// TIA Portal V17 export
// export: Created 2025-03-05T08:03:01.8804451Z, ExportSetting WithDefaults, DisplayName Totally Integrated Automation Portal, DisplayVersion V17 Update 8, DisplayName TIA Portal Openness, DisplayVersion V17 Update 8, DisplayName TIA Portal Version Control Interface, DisplayVersion V17, DisplayName SINAMICS Startdrive Advanced, DisplayVersion V17 SP2, DisplayName SINAMICS Startdrive G110M, G120, G120C, G120D, G120P, G115D, DisplayVersion V17 SP2, DisplayName SINAMICS Startdrive G130, G150, S120, S150, SINAMICS MV, S210, DisplayVersion V17 SP2, DisplayName STEP 7 Professional, DisplayVersion V17 Update 8, DisplayName SINUMERIK ONE STEP 7 Toolbox, DisplayVersion V17 Update 12, DisplayName SINUMERIK 840D sl STEP 7 Toolbox, DisplayVersion V17 Update 12, DisplayName STEP 7 Safety, DisplayVersion V17 Update 6, DisplayName WinCC Advanced, DisplayVersion V17 Update 8
FUNCTION "FC21011_POWDER_FEEDER_GENERAL" : Void   // FC21011, LAD
TITLE = FC21011 POWDER FEEDER GENERAL
{ S7_Optimized_Access := 'TRUE' }
VERSION : 0.1
// stored: AutoNumber false, IsIECCheckEnabled false, SetENOAutomatically false, UDAEnableTagReadback false
BEGIN

REGION Network 1: /////_UNIT_01_/////
END_REGION

REGION Network 2: CALL FB21011 POWDER FEEDER 1 GENERAL UNIT 01
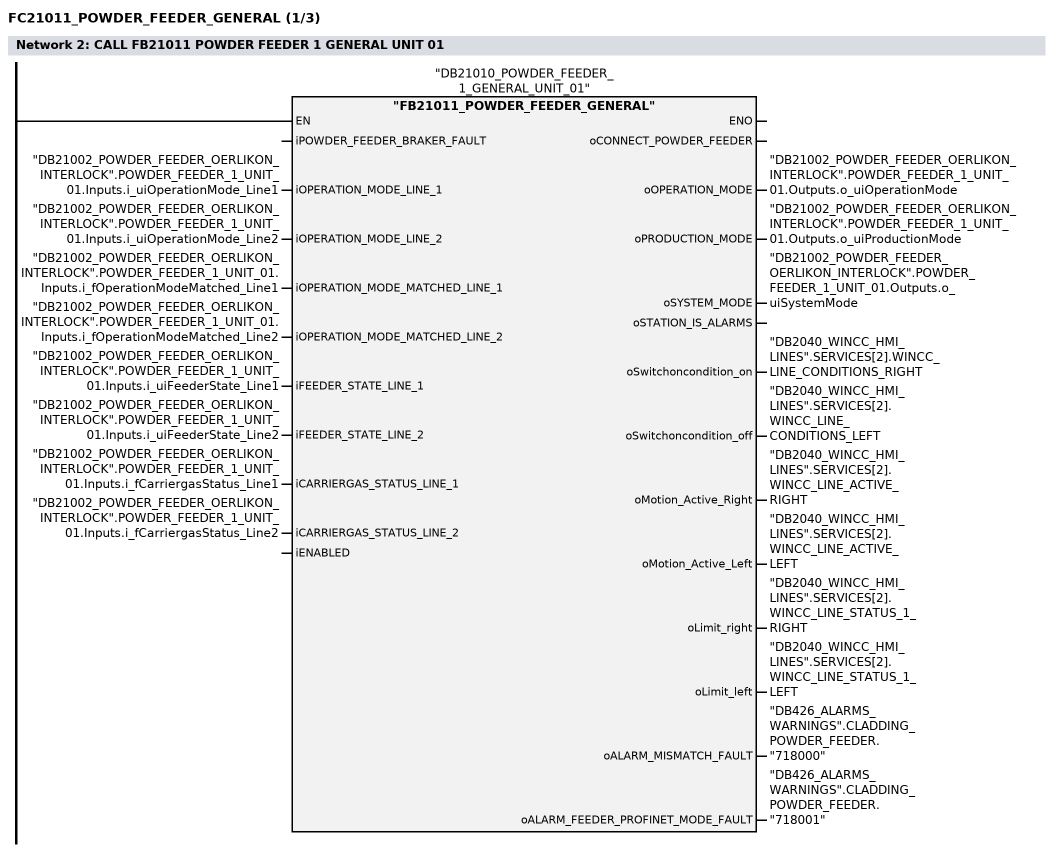
   RUNG wire#powerrail
      "DB21010_POWDER_FEEDER_1_GENERAL_UNIT_01"(iPOWDER_FEEDER_BRAKER_FAULT :=, iOPERATION_MODE_LINE_1 := "DB21002_POWDER_FEEDER_OERLIKON_INTERLOCK".POWDER_FEEDER_1_UNIT_01.Inputs.i_uiOperationMode_Line1, iOPERATION_MODE_LINE_2 := "DB21002_POWDER_FEEDER_OERLIKON_INTERLOCK".POWDER_FEEDER_1_UNIT_01.Inputs.i_uiOperationMode_Line2, iOPERATION_MODE_MATCHED_LINE_1 := "DB21002_POWDER_FEEDER_OERLIKON_INTERLOCK".POWDER_FEEDER_1_UNIT_01.Inputs.i_fOperationModeMatched_Line1, iOPERATION_MODE_MATCHED_LINE_2 := "DB21002_POWDER_FEEDER_OERLIKON_INTERLOCK".POWDER_FEEDER_1_UNIT_01.Inputs.i_fOperationModeMatched_Line2, iFEEDER_STATE_LINE_1 := "DB21002_POWDER_FEEDER_OERLIKON_INTERLOCK".POWDER_FEEDER_1_UNIT_01.Inputs.i_uiFeederState_Line1, iFEEDER_STATE_LINE_2 := "DB21002_POWDER_FEEDER_OERLIKON_INTERLOCK".POWDER_FEEDER_1_UNIT_01.Inputs.i_uiFeederState_Line2, iCARRIERGAS_STATUS_LINE_1 := "DB21002_POWDER_FEEDER_OERLIKON_INTERLOCK".POWDER_FEEDER_1_UNIT_01.Inputs.i_fCarriergasStatus_Line1, iCARRIERGAS_STATUS_LINE_2 := "DB21002_POWDER_FEEDER_OERLIKON_INTERLOCK".POWDER_FEEDER_1_UNIT_01.Inputs.i_fCarriergasStatus_Line2, iENABLED :=, oCONNECT_POWDER_FEEDER =>, oOPERATION_MODE => "DB21002_POWDER_FEEDER_OERLIKON_INTERLOCK".POWDER_FEEDER_1_UNIT_01.Outputs.o_uiOperationMode, oPRODUCTION_MODE => "DB21002_POWDER_FEEDER_OERLIKON_INTERLOCK".POWDER_FEEDER_1_UNIT_01.Outputs.o_uiProductionMode, oSYSTEM_MODE => "DB21002_POWDER_FEEDER_OERLIKON_INTERLOCK".POWDER_FEEDER_1_UNIT_01.Outputs.o_uiSystemMode, oSTATION_IS_ALARMS =>, oSwitchoncondition_on => "DB2040_WINCC_HMI_LINES".SERVICES[2].WINCC_LINE_CONDITIONS_RIGHT, oSwitchoncondition_off => "DB2040_WINCC_HMI_LINES".SERVICES[2].WINCC_LINE_CONDITIONS_LEFT, oMotion_Active_Right => "DB2040_WINCC_HMI_LINES".SERVICES[2].WINCC_LINE_ACTIVE_RIGHT, oMotion_Active_Left => "DB2040_WINCC_HMI_LINES".SERVICES[2].WINCC_LINE_ACTIVE_LEFT, oLimit_right => "DB2040_WINCC_HMI_LINES".SERVICES[2].WINCC_LINE_STATUS_1_RIGHT, oLimit_left => "DB2040_WINCC_HMI_LINES".SERVICES[2].WINCC_LINE_STATUS_1_LEFT, oALARM_MISMATCH_FAULT => "DB426_ALARMS_WARNINGS".CLADDING_POWDER_FEEDER."718000", oALARM_FEEDER_PROFINET_MODE_FAULT => "DB426_ALARMS_WARNINGS".CLADDING_POWDER_FEEDER."718001")
   END_RUNG
   // the same network as SCL:
   "DB21010_POWDER_FEEDER_1_GENERAL_UNIT_01"(iOPERATION_MODE_LINE_1 := "DB21002_POWDER_FEEDER_OERLIKON_INTERLOCK".POWDER_FEEDER_1_UNIT_01.Inputs.i_uiOperationMode_Line1,   // "FB21011_POWDER_FEEDER_GENERAL"
                           iOPERATION_MODE_LINE_2 := "DB21002_POWDER_FEEDER_OERLIKON_INTERLOCK".POWDER_FEEDER_1_UNIT_01.Inputs.i_uiOperationMode_Line2,
                           iOPERATION_MODE_MATCHED_LINE_1 := "DB21002_POWDER_FEEDER_OERLIKON_INTERLOCK".POWDER_FEEDER_1_UNIT_01.Inputs.i_fOperationModeMatched_Line1,
                           iOPERATION_MODE_MATCHED_LINE_2 := "DB21002_POWDER_FEEDER_OERLIKON_INTERLOCK".POWDER_FEEDER_1_UNIT_01.Inputs.i_fOperationModeMatched_Line2,
                           iFEEDER_STATE_LINE_1 := "DB21002_POWDER_FEEDER_OERLIKON_INTERLOCK".POWDER_FEEDER_1_UNIT_01.Inputs.i_uiFeederState_Line1,
                           iFEEDER_STATE_LINE_2 := "DB21002_POWDER_FEEDER_OERLIKON_INTERLOCK".POWDER_FEEDER_1_UNIT_01.Inputs.i_uiFeederState_Line2,
                           iCARRIERGAS_STATUS_LINE_1 := "DB21002_POWDER_FEEDER_OERLIKON_INTERLOCK".POWDER_FEEDER_1_UNIT_01.Inputs.i_fCarriergasStatus_Line1,
                           iCARRIERGAS_STATUS_LINE_2 := "DB21002_POWDER_FEEDER_OERLIKON_INTERLOCK".POWDER_FEEDER_1_UNIT_01.Inputs.i_fCarriergasStatus_Line2,
                           oOPERATION_MODE => "DB21002_POWDER_FEEDER_OERLIKON_INTERLOCK".POWDER_FEEDER_1_UNIT_01.Outputs.o_uiOperationMode,
                           oPRODUCTION_MODE => "DB21002_POWDER_FEEDER_OERLIKON_INTERLOCK".POWDER_FEEDER_1_UNIT_01.Outputs.o_uiProductionMode,
                           oSYSTEM_MODE => "DB21002_POWDER_FEEDER_OERLIKON_INTERLOCK".POWDER_FEEDER_1_UNIT_01.Outputs.o_uiSystemMode,
                           oSwitchoncondition_on => "DB2040_WINCC_HMI_LINES".SERVICES[2].WINCC_LINE_CONDITIONS_RIGHT,
                           oSwitchoncondition_off => "DB2040_WINCC_HMI_LINES".SERVICES[2].WINCC_LINE_CONDITIONS_LEFT,
                           oMotion_Active_Right => "DB2040_WINCC_HMI_LINES".SERVICES[2].WINCC_LINE_ACTIVE_RIGHT,
                           oMotion_Active_Left => "DB2040_WINCC_HMI_LINES".SERVICES[2].WINCC_LINE_ACTIVE_LEFT,
                           oLimit_right => "DB2040_WINCC_HMI_LINES".SERVICES[2].WINCC_LINE_STATUS_1_RIGHT,
                           oLimit_left => "DB2040_WINCC_HMI_LINES".SERVICES[2].WINCC_LINE_STATUS_1_LEFT,
                           oALARM_MISMATCH_FAULT => "DB426_ALARMS_WARNINGS".CLADDING_POWDER_FEEDER."718000",
                           oALARM_FEEDER_PROFINET_MODE_FAULT => "DB426_ALARMS_WARNINGS".CLADDING_POWDER_FEEDER."718001");
END_REGION

REGION Network 3: /////_UNIT_02_/////
END_REGION

REGION Network 4: CALL FB21011 POWDER FEEDER 1 GENERAL UNIT 02
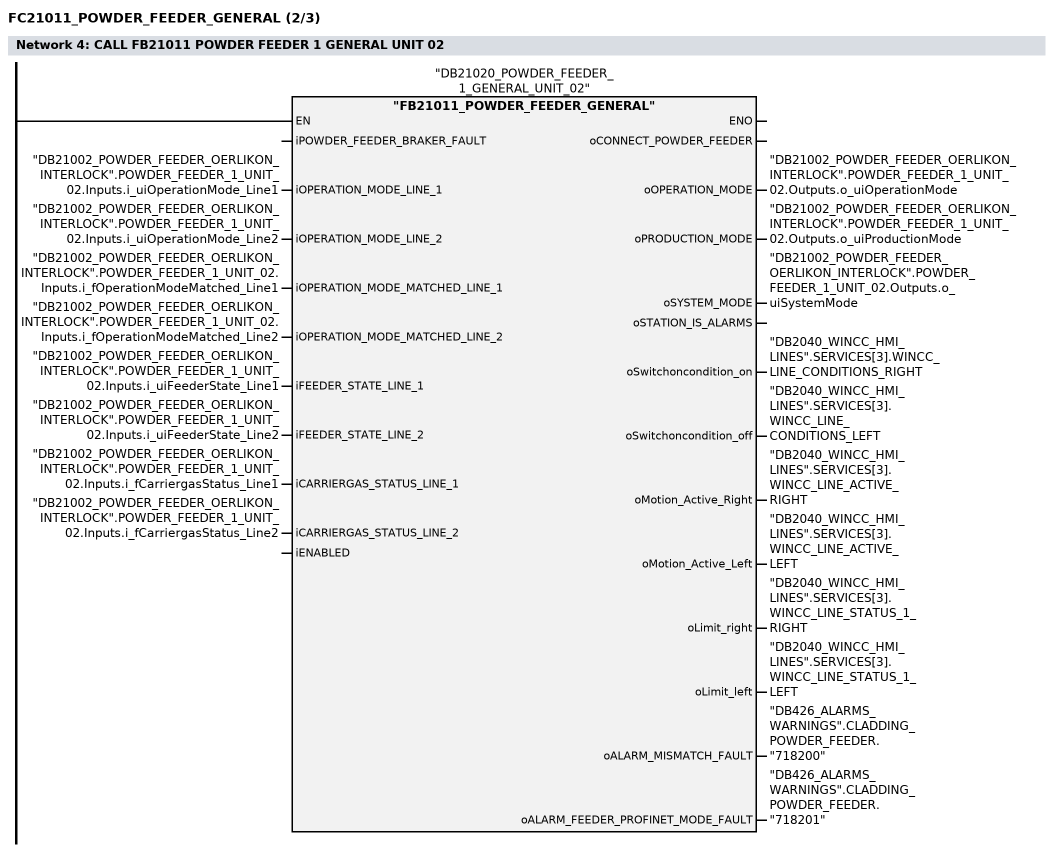
   RUNG wire#powerrail
      "DB21020_POWDER_FEEDER_1_GENERAL_UNIT_02"(iPOWDER_FEEDER_BRAKER_FAULT :=, iOPERATION_MODE_LINE_1 := "DB21002_POWDER_FEEDER_OERLIKON_INTERLOCK".POWDER_FEEDER_1_UNIT_02.Inputs.i_uiOperationMode_Line1, iOPERATION_MODE_LINE_2 := "DB21002_POWDER_FEEDER_OERLIKON_INTERLOCK".POWDER_FEEDER_1_UNIT_02.Inputs.i_uiOperationMode_Line2, iOPERATION_MODE_MATCHED_LINE_1 := "DB21002_POWDER_FEEDER_OERLIKON_INTERLOCK".POWDER_FEEDER_1_UNIT_02.Inputs.i_fOperationModeMatched_Line1, iOPERATION_MODE_MATCHED_LINE_2 := "DB21002_POWDER_FEEDER_OERLIKON_INTERLOCK".POWDER_FEEDER_1_UNIT_02.Inputs.i_fOperationModeMatched_Line2, iFEEDER_STATE_LINE_1 := "DB21002_POWDER_FEEDER_OERLIKON_INTERLOCK".POWDER_FEEDER_1_UNIT_02.Inputs.i_uiFeederState_Line1, iFEEDER_STATE_LINE_2 := "DB21002_POWDER_FEEDER_OERLIKON_INTERLOCK".POWDER_FEEDER_1_UNIT_02.Inputs.i_uiFeederState_Line2, iCARRIERGAS_STATUS_LINE_1 := "DB21002_POWDER_FEEDER_OERLIKON_INTERLOCK".POWDER_FEEDER_1_UNIT_02.Inputs.i_fCarriergasStatus_Line1, iCARRIERGAS_STATUS_LINE_2 := "DB21002_POWDER_FEEDER_OERLIKON_INTERLOCK".POWDER_FEEDER_1_UNIT_02.Inputs.i_fCarriergasStatus_Line2, iENABLED :=, oCONNECT_POWDER_FEEDER =>, oOPERATION_MODE => "DB21002_POWDER_FEEDER_OERLIKON_INTERLOCK".POWDER_FEEDER_1_UNIT_02.Outputs.o_uiOperationMode, oPRODUCTION_MODE => "DB21002_POWDER_FEEDER_OERLIKON_INTERLOCK".POWDER_FEEDER_1_UNIT_02.Outputs.o_uiProductionMode, oSYSTEM_MODE => "DB21002_POWDER_FEEDER_OERLIKON_INTERLOCK".POWDER_FEEDER_1_UNIT_02.Outputs.o_uiSystemMode, oSTATION_IS_ALARMS =>, oSwitchoncondition_on => "DB2040_WINCC_HMI_LINES".SERVICES[3].WINCC_LINE_CONDITIONS_RIGHT, oSwitchoncondition_off => "DB2040_WINCC_HMI_LINES".SERVICES[3].WINCC_LINE_CONDITIONS_LEFT, oMotion_Active_Right => "DB2040_WINCC_HMI_LINES".SERVICES[3].WINCC_LINE_ACTIVE_RIGHT, oMotion_Active_Left => "DB2040_WINCC_HMI_LINES".SERVICES[3].WINCC_LINE_ACTIVE_LEFT, oLimit_right => "DB2040_WINCC_HMI_LINES".SERVICES[3].WINCC_LINE_STATUS_1_RIGHT, oLimit_left => "DB2040_WINCC_HMI_LINES".SERVICES[3].WINCC_LINE_STATUS_1_LEFT, oALARM_MISMATCH_FAULT => "DB426_ALARMS_WARNINGS".CLADDING_POWDER_FEEDER."718200", oALARM_FEEDER_PROFINET_MODE_FAULT => "DB426_ALARMS_WARNINGS".CLADDING_POWDER_FEEDER."718201")
   END_RUNG
   // the same network as SCL:
   "DB21020_POWDER_FEEDER_1_GENERAL_UNIT_02"(iOPERATION_MODE_LINE_1 := "DB21002_POWDER_FEEDER_OERLIKON_INTERLOCK".POWDER_FEEDER_1_UNIT_02.Inputs.i_uiOperationMode_Line1,   // "FB21011_POWDER_FEEDER_GENERAL"
                           iOPERATION_MODE_LINE_2 := "DB21002_POWDER_FEEDER_OERLIKON_INTERLOCK".POWDER_FEEDER_1_UNIT_02.Inputs.i_uiOperationMode_Line2,
                           iOPERATION_MODE_MATCHED_LINE_1 := "DB21002_POWDER_FEEDER_OERLIKON_INTERLOCK".POWDER_FEEDER_1_UNIT_02.Inputs.i_fOperationModeMatched_Line1,
                           iOPERATION_MODE_MATCHED_LINE_2 := "DB21002_POWDER_FEEDER_OERLIKON_INTERLOCK".POWDER_FEEDER_1_UNIT_02.Inputs.i_fOperationModeMatched_Line2,
                           iFEEDER_STATE_LINE_1 := "DB21002_POWDER_FEEDER_OERLIKON_INTERLOCK".POWDER_FEEDER_1_UNIT_02.Inputs.i_uiFeederState_Line1,
                           iFEEDER_STATE_LINE_2 := "DB21002_POWDER_FEEDER_OERLIKON_INTERLOCK".POWDER_FEEDER_1_UNIT_02.Inputs.i_uiFeederState_Line2,
                           iCARRIERGAS_STATUS_LINE_1 := "DB21002_POWDER_FEEDER_OERLIKON_INTERLOCK".POWDER_FEEDER_1_UNIT_02.Inputs.i_fCarriergasStatus_Line1,
                           iCARRIERGAS_STATUS_LINE_2 := "DB21002_POWDER_FEEDER_OERLIKON_INTERLOCK".POWDER_FEEDER_1_UNIT_02.Inputs.i_fCarriergasStatus_Line2,
                           oOPERATION_MODE => "DB21002_POWDER_FEEDER_OERLIKON_INTERLOCK".POWDER_FEEDER_1_UNIT_02.Outputs.o_uiOperationMode,
                           oPRODUCTION_MODE => "DB21002_POWDER_FEEDER_OERLIKON_INTERLOCK".POWDER_FEEDER_1_UNIT_02.Outputs.o_uiProductionMode,
                           oSYSTEM_MODE => "DB21002_POWDER_FEEDER_OERLIKON_INTERLOCK".POWDER_FEEDER_1_UNIT_02.Outputs.o_uiSystemMode,
                           oSwitchoncondition_on => "DB2040_WINCC_HMI_LINES".SERVICES[3].WINCC_LINE_CONDITIONS_RIGHT,
                           oSwitchoncondition_off => "DB2040_WINCC_HMI_LINES".SERVICES[3].WINCC_LINE_CONDITIONS_LEFT,
                           oMotion_Active_Right => "DB2040_WINCC_HMI_LINES".SERVICES[3].WINCC_LINE_ACTIVE_RIGHT,
                           oMotion_Active_Left => "DB2040_WINCC_HMI_LINES".SERVICES[3].WINCC_LINE_ACTIVE_LEFT,
                           oLimit_right => "DB2040_WINCC_HMI_LINES".SERVICES[3].WINCC_LINE_STATUS_1_RIGHT,
                           oLimit_left => "DB2040_WINCC_HMI_LINES".SERVICES[3].WINCC_LINE_STATUS_1_LEFT,
                           oALARM_MISMATCH_FAULT => "DB426_ALARMS_WARNINGS".CLADDING_POWDER_FEEDER."718200",
                           oALARM_FEEDER_PROFINET_MODE_FAULT => "DB426_ALARMS_WARNINGS".CLADDING_POWDER_FEEDER."718201");
END_REGION

REGION Network 5: CALL FB21011 POWDER FEEDER 2 GENERAL UNIT 02
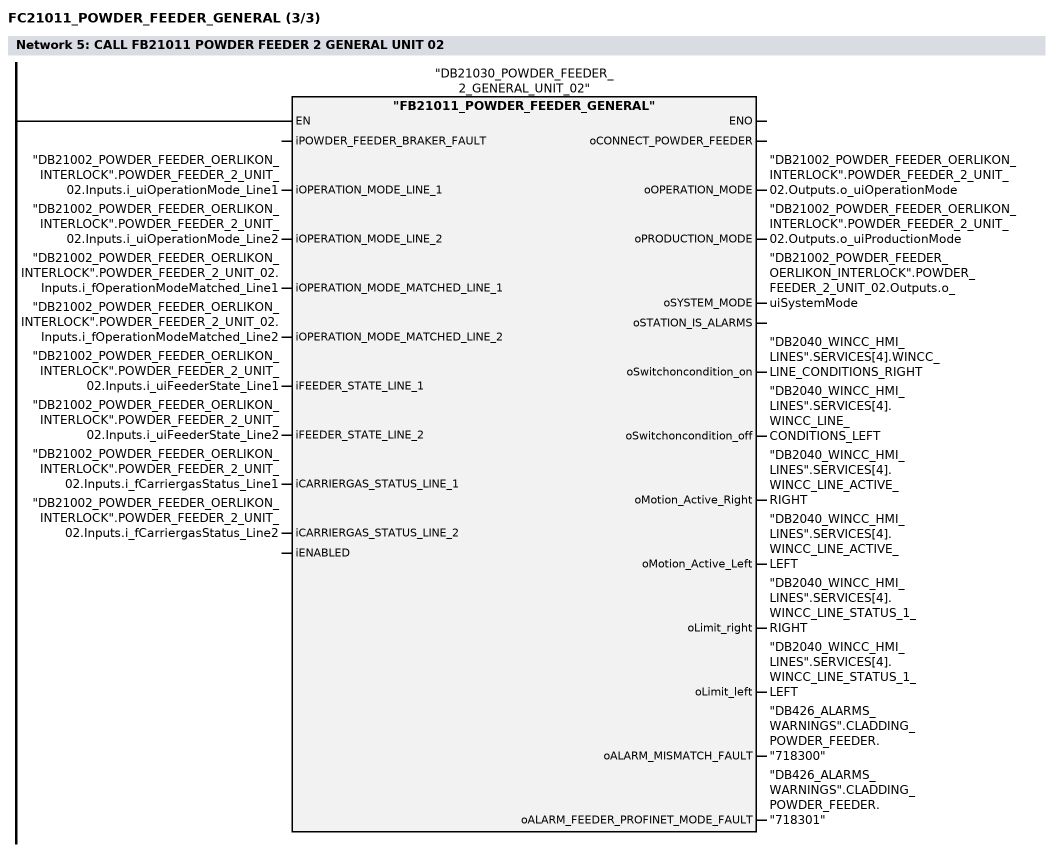
   RUNG wire#powerrail
      "DB21030_POWDER_FEEDER_2_GENERAL_UNIT_02"(iPOWDER_FEEDER_BRAKER_FAULT :=, iOPERATION_MODE_LINE_1 := "DB21002_POWDER_FEEDER_OERLIKON_INTERLOCK".POWDER_FEEDER_2_UNIT_02.Inputs.i_uiOperationMode_Line1, iOPERATION_MODE_LINE_2 := "DB21002_POWDER_FEEDER_OERLIKON_INTERLOCK".POWDER_FEEDER_2_UNIT_02.Inputs.i_uiOperationMode_Line2, iOPERATION_MODE_MATCHED_LINE_1 := "DB21002_POWDER_FEEDER_OERLIKON_INTERLOCK".POWDER_FEEDER_2_UNIT_02.Inputs.i_fOperationModeMatched_Line1, iOPERATION_MODE_MATCHED_LINE_2 := "DB21002_POWDER_FEEDER_OERLIKON_INTERLOCK".POWDER_FEEDER_2_UNIT_02.Inputs.i_fOperationModeMatched_Line2, iFEEDER_STATE_LINE_1 := "DB21002_POWDER_FEEDER_OERLIKON_INTERLOCK".POWDER_FEEDER_2_UNIT_02.Inputs.i_uiFeederState_Line1, iFEEDER_STATE_LINE_2 := "DB21002_POWDER_FEEDER_OERLIKON_INTERLOCK".POWDER_FEEDER_2_UNIT_02.Inputs.i_uiFeederState_Line2, iCARRIERGAS_STATUS_LINE_1 := "DB21002_POWDER_FEEDER_OERLIKON_INTERLOCK".POWDER_FEEDER_2_UNIT_02.Inputs.i_fCarriergasStatus_Line1, iCARRIERGAS_STATUS_LINE_2 := "DB21002_POWDER_FEEDER_OERLIKON_INTERLOCK".POWDER_FEEDER_2_UNIT_02.Inputs.i_fCarriergasStatus_Line2, iENABLED :=, oCONNECT_POWDER_FEEDER =>, oOPERATION_MODE => "DB21002_POWDER_FEEDER_OERLIKON_INTERLOCK".POWDER_FEEDER_2_UNIT_02.Outputs.o_uiOperationMode, oPRODUCTION_MODE => "DB21002_POWDER_FEEDER_OERLIKON_INTERLOCK".POWDER_FEEDER_2_UNIT_02.Outputs.o_uiProductionMode, oSYSTEM_MODE => "DB21002_POWDER_FEEDER_OERLIKON_INTERLOCK".POWDER_FEEDER_2_UNIT_02.Outputs.o_uiSystemMode, oSTATION_IS_ALARMS =>, oSwitchoncondition_on => "DB2040_WINCC_HMI_LINES".SERVICES[4].WINCC_LINE_CONDITIONS_RIGHT, oSwitchoncondition_off => "DB2040_WINCC_HMI_LINES".SERVICES[4].WINCC_LINE_CONDITIONS_LEFT, oMotion_Active_Right => "DB2040_WINCC_HMI_LINES".SERVICES[4].WINCC_LINE_ACTIVE_RIGHT, oMotion_Active_Left => "DB2040_WINCC_HMI_LINES".SERVICES[4].WINCC_LINE_ACTIVE_LEFT, oLimit_right => "DB2040_WINCC_HMI_LINES".SERVICES[4].WINCC_LINE_STATUS_1_RIGHT, oLimit_left => "DB2040_WINCC_HMI_LINES".SERVICES[4].WINCC_LINE_STATUS_1_LEFT, oALARM_MISMATCH_FAULT => "DB426_ALARMS_WARNINGS".CLADDING_POWDER_FEEDER."718300", oALARM_FEEDER_PROFINET_MODE_FAULT => "DB426_ALARMS_WARNINGS".CLADDING_POWDER_FEEDER."718301")
   END_RUNG
   // the same network as SCL:
   "DB21030_POWDER_FEEDER_2_GENERAL_UNIT_02"(iOPERATION_MODE_LINE_1 := "DB21002_POWDER_FEEDER_OERLIKON_INTERLOCK".POWDER_FEEDER_2_UNIT_02.Inputs.i_uiOperationMode_Line1,   // "FB21011_POWDER_FEEDER_GENERAL"
                           iOPERATION_MODE_LINE_2 := "DB21002_POWDER_FEEDER_OERLIKON_INTERLOCK".POWDER_FEEDER_2_UNIT_02.Inputs.i_uiOperationMode_Line2,
                           iOPERATION_MODE_MATCHED_LINE_1 := "DB21002_POWDER_FEEDER_OERLIKON_INTERLOCK".POWDER_FEEDER_2_UNIT_02.Inputs.i_fOperationModeMatched_Line1,
                           iOPERATION_MODE_MATCHED_LINE_2 := "DB21002_POWDER_FEEDER_OERLIKON_INTERLOCK".POWDER_FEEDER_2_UNIT_02.Inputs.i_fOperationModeMatched_Line2,
                           iFEEDER_STATE_LINE_1 := "DB21002_POWDER_FEEDER_OERLIKON_INTERLOCK".POWDER_FEEDER_2_UNIT_02.Inputs.i_uiFeederState_Line1,
                           iFEEDER_STATE_LINE_2 := "DB21002_POWDER_FEEDER_OERLIKON_INTERLOCK".POWDER_FEEDER_2_UNIT_02.Inputs.i_uiFeederState_Line2,
                           iCARRIERGAS_STATUS_LINE_1 := "DB21002_POWDER_FEEDER_OERLIKON_INTERLOCK".POWDER_FEEDER_2_UNIT_02.Inputs.i_fCarriergasStatus_Line1,
                           iCARRIERGAS_STATUS_LINE_2 := "DB21002_POWDER_FEEDER_OERLIKON_INTERLOCK".POWDER_FEEDER_2_UNIT_02.Inputs.i_fCarriergasStatus_Line2,
                           oOPERATION_MODE => "DB21002_POWDER_FEEDER_OERLIKON_INTERLOCK".POWDER_FEEDER_2_UNIT_02.Outputs.o_uiOperationMode,
                           oPRODUCTION_MODE => "DB21002_POWDER_FEEDER_OERLIKON_INTERLOCK".POWDER_FEEDER_2_UNIT_02.Outputs.o_uiProductionMode,
                           oSYSTEM_MODE => "DB21002_POWDER_FEEDER_OERLIKON_INTERLOCK".POWDER_FEEDER_2_UNIT_02.Outputs.o_uiSystemMode,
                           oSwitchoncondition_on => "DB2040_WINCC_HMI_LINES".SERVICES[4].WINCC_LINE_CONDITIONS_RIGHT,
                           oSwitchoncondition_off => "DB2040_WINCC_HMI_LINES".SERVICES[4].WINCC_LINE_CONDITIONS_LEFT,
                           oMotion_Active_Right => "DB2040_WINCC_HMI_LINES".SERVICES[4].WINCC_LINE_ACTIVE_RIGHT,
                           oMotion_Active_Left => "DB2040_WINCC_HMI_LINES".SERVICES[4].WINCC_LINE_ACTIVE_LEFT,
                           oLimit_right => "DB2040_WINCC_HMI_LINES".SERVICES[4].WINCC_LINE_STATUS_1_RIGHT,
                           oLimit_left => "DB2040_WINCC_HMI_LINES".SERVICES[4].WINCC_LINE_STATUS_1_LEFT,
                           oALARM_MISMATCH_FAULT => "DB426_ALARMS_WARNINGS".CLADDING_POWDER_FEEDER."718300",
                           oALARM_FEEDER_PROFINET_MODE_FAULT => "DB426_ALARMS_WARNINGS".CLADDING_POWDER_FEEDER."718301");
END_REGION
END_FUNCTION
